// TIA Portal V19 export
TYPE "MES_Msg_Receive_Topic1xx_Err"
// stored: Access Published
   STRUCT
      Recive_MSG100 { ExternalAccessible := 'False'; ExternalVisible := 'False'; ExternalWritable := 'False'} : "MES_Err_&_Msg";
      Recive_MSG130 { ExternalAccessible := 'False'; ExternalVisible := 'False'; ExternalWritable := 'False'} : "MES_Err_&_Msg";
      Recive_MSG140 { ExternalAccessible := 'False'; ExternalVisible := 'False'; ExternalWritable := 'False'} : "MES_Err_&_Msg";
      Recive_MSG142 { ExternalAccessible := 'False'; ExternalVisible := 'False'; ExternalWritable := 'False'} : "MES_Err_&_Msg";
      Send_MSG131_Follow_MSG130 { ExternalAccessible := 'False'; ExternalVisible := 'False'; ExternalWritable := 'False'} : "MES_Err_&_Msg";
      Send_MSG141_Follow_MSG140 { ExternalAccessible := 'False'; ExternalVisible := 'False'; ExternalWritable := 'False'} : "MES_Err_&_Msg";
      Send_MSG143_Follow_MSG142 { ExternalAccessible := 'False'; ExternalVisible := 'False'; ExternalWritable := 'False'} : "MES_Err_&_Msg";
      Send_MSG144_Follow_MSG142 { ExternalAccessible := 'False'; ExternalVisible := 'False'; ExternalWritable := 'False'} : "MES_Err_&_Msg";
      Send_MSG145_Follow_MSG142 { ExternalAccessible := 'False'; ExternalVisible := 'False'; ExternalWritable := 'False'} : "MES_Err_&_Msg";
   END_STRUCT;
END_TYPE
